TYPE ST_HaveDUTState :
STRUCT
	haveDUT:BOOL;
	DutCheckDone:BOOL;
	DutCheckRuslut:BOOL;
END_STRUCT
END_TYPE

(* stored: Version 1.1.0.1, ProductVersion 3.1.4024.4
   DUT ST_HaveDUTState: Id {7a50f21d-afb3-401b-9506-62dc0c691cf7} *)
